// TwinCAT 3 PLC project TcSequencer
// Title: TcSequencer
// Company: Loupe
// ProjectVersion: 0.0.5
// ProgramVersion: 3.1.4024.0
// libraries:
//   Tc2_Standard, * (Beckhoff Automation GmbH)
//   Tc2_System, * (Beckhoff Automation GmbH)
//   Tc3_Module, * (Beckhoff Automation GmbH)
//   TcCommando, * (Loupe)
//   TcPluginFramework, * (Loupe)
//   TcUnit, * (www.tcunit.org)
// project tree:
//   DUTs/ SequenceCommand.TcDUT, SequenceType.TcDUT, SEQUENCE_STEP.TcTLEO
//   Example/ ExampleProg1.TcPOU, ExampleSeq1.TcPOU, IMOCK_EM.TcIO, Mock_EM.TcPOU
//   Interfaces/ ISequence.TcIO, IStepManager.TcIO
//   / PlcTask.TcTTO
//   POUs/ Sequencer.TcPOU, StepManagerBasic.TcPOU
//   Test/ Sequencer_Test.TcPOU, StepManagerBasic_Test.TcPOU, TESTPRG.TcPOU
// real-time tasks:
//   TASK PlcTask: cycle T#10ms, priority 20, ADS port 350

CONFIGURATION TcSequencer
    RESOURCE PLC ON TwinCAT3
        TASK PlcTask(INTERVAL := T#10ms, PRIORITY := 20);
        PROGRAM TESTPRG WITH PlcTask : TESTPRG;
        PROGRAM ExampleProg1 WITH PlcTask : ExampleProg1;
    END_RESOURCE
END_CONFIGURATION

// ---- DUTs/SequenceCommand.TcDUT
TYPE SequenceCommand :
STRUCT
	Start : PLCopenCommand;
	Stop : PLCopenCommand;
END_STRUCT
END_TYPE

// ---- DUTs/SequenceType.TcDUT
TYPE
    SequenceType :
    STRUCT
        startStep : ENUM; //The step when doStep was called
        currentStep : ENUM;
        lastRequestNumber : DINT;

        onEntry : BOOL;
        onExit : BOOL;

        statusChecked : BOOL;
        isDone : BOOL;
        isAbort : BOOL;
        isError : BOOL;

        errorHandled : BOOL;

    END_STRUCT
END_TYPE

// ---- DUTs/SEQUENCE_STEP.TcTLEO
{attribute 'qualified_only'}
TYPE SEQUENCE_STEP :
(
	STEP_ERROR := -3,
	NO_STEP_CHANGE := -2,
	NO_STEP := -1,
	IDLE_STEP := 0,
	START_STEP := 1
);
END_TYPE
//  STEP_ERROR = '-3'
//  NO_STEP_CHANGE = '-2'
//  NO_STEP = '-1'

// ---- Example/IMOCK_EM.TcIO
INTERFACE IMOCK_EM


METHOD MoveDown : BOOL
VAR_INPUT
  Status : IPLCopenCall;
END_VAR
END_METHOD


METHOD MoveUp : BOOL
VAR_INPUT
  Status : IPLCopenCall;
END_VAR
END_METHOD

END_INTERFACE

// ---- Interfaces/ISequence.TcIO
INTERFACE ISequence
// Copyright (c) 2024 Loupe (https://loupe.team), provided under the MIT License.

{attribute 'monitoring' := 'call'}
PROPERTY CurrentStep : ENUM
GET
END_GET
END_PROPERTY

METHOD DoStep : ENUM
VAR
END_VAR
END_METHOD

METHOD OnAbort : BOOL
VAR_INPUT
    nextStep : ENUM;
END_VAR
END_METHOD

METHOD OnEntry : BOOL
VAR_INPUT
END_VAR
END_METHOD

METHOD OnError : BOOL
VAR_INPUT
    nextStep : ENUM;
END_VAR
END_METHOD

METHOD OnExit : BOOL
VAR_INPUT
END_VAR
END_METHOD

METHOD OnFailure : BOOL
VAR_INPUT
    nextStep : ENUM;
END_VAR
END_METHOD

METHOD OnSuccess : BOOL
VAR_INPUT
    nextStep : ENUM;
END_VAR
END_METHOD

METHOD RequestStep : BOOL
VAR_INPUT
    nextStep : ENUM;
END_VAR
END_METHOD

METHOD RequestStepClear : BOOL
VAR_INPUT
    nextStep : ENUM;
END_VAR
END_METHOD

METHOD SequenceAbort : BOOL
VAR_INPUT
    ErrorCode : DINT;
    ErrorMessage : STRING;
END_VAR
END_METHOD

METHOD SequenceComplete : BOOL
VAR_INPUT
END_VAR
END_METHOD

METHOD SequenceError : BOOL
VAR_INPUT
    ErrorCode : INT;
    ErrorMessage : STRING;
END_VAR
END_METHOD

METHOD SetStepManager : BOOL
VAR_INPUT
	manager : IStepManager;
END_VAR
END_METHOD

METHOD StartSequence : BOOL
VAR_INPUT
	Status : IPLCopenCaller;
END_VAR
END_METHOD

END_INTERFACE

// ---- Interfaces/IStepManager.TcIO
INTERFACE IStepManager
// Copyright (c) 2024 Loupe (https://loupe.team), provided under the MIT License.

PROPERTY CurrentStepImpl : ENUM
GET
END_GET
END_PROPERTY

PROPERTY RequestNumberImpl : DINT
GET
END_GET
END_PROPERTY

METHOD RequestStepImpl : BOOL
VAR_INPUT
    nextStep : ENUM;
END_VAR
END_METHOD

METHOD ResetImpl : BOOL
VAR_INPUT
END_VAR
END_METHOD

METHOD SequenceCompleteImpl : BOOL
VAR_INPUT
END_VAR
END_METHOD

METHOD SequenceErrorImpl : BOOL
VAR_INPUT
    ErrorCode : INT;
    ErrorMessage : STRING;
END_VAR
END_METHOD

END_INTERFACE

// ---- Test/TESTPRG.TcPOU
{attribute 'no-analysis'}
PROGRAM TESTPRG
VAR
    sequencerTest : Sequencer_Test;
    stepManagerTest : StepManagerBasic_Test;
END_VAR

// Copyright (c) 2024 Loupe (https://loupe.team), provided under the MIT License.

TcUnit.RUN();

END_PROGRAM

// ---- Test/Sequencer_Test.TcPOU
FUNCTION_BLOCK Sequencer_Test EXTENDS FB_TestSuite
VAR_INPUT
END_VAR
VAR_OUTPUT
END_VAR
VAR
END_VAR

// Copyright (c) 2024 Loupe (https://loupe.team), provided under the MIT License.

OnAbort();
OnEntry();
CurrentAndRequestStep();

{attribute 'no-analysis'}
METHOD CurrentAndRequestStep
VAR
    sequencer : Sequencer(0);
    Command : PLCopenCommand();
    step : UDINT;
END_VAR
// Copyright (c) 2024 Loupe (https://loupe.team), provided under the MIT License.

(*STweep.Disable*)

TEST('CurrentAndRequestStep');
	AssertEquals_UDINT(Expected := 0, Actual := sequencer.CurrentStep, Message := 'Current step shall default to 0');
	
	step := 2;
	sequencer.RequestStep(step);
	AssertEquals_UDINT(Expected := step, Actual := sequencer.CurrentStep, Message := 'Current step expected to be updated');
	
	step := 3;
	sequencer.RequestStepClear(step);
	AssertEquals_UDINT(Expected := step, Actual := sequencer.CurrentStep, Message := 'Current step expected to be updated');
TEST_FINISHED();
END_METHOD

{attribute 'no-analysis'}
METHOD OnAbort
VAR
    sequencer : Sequencer(0);
    outputVal : BOOL;
	Command : PLCopenCommand;
END_VAR
// Copyright (c) 2024 Loupe (https://loupe.team), provided under the MIT License.

(*STweep.Disable*)

TEST('SequenceOnAbort');
	sequencer.RequestStep(1);
	sequencer.DoStep();
	sequencer.Start(Command);
	Command.Execute := TRUE;
	IF sequencer.OnAbort(-1) THEN
		outputVal := sequencer.SequenceAbort(1, 'Command aborted');
	END_IF
	AssertTrue(Condition := outputVal, Message := 'Abort should be true');
TEST_FINISHED();
END_METHOD

{attribute 'no-analysis'}
METHOD OnEntry
VAR_INPUT
END_VAR

VAR
    sequencer : Sequencer(0);
    outputVal : BOOL;
END_VAR
// Copyright (c) 2024 Loupe (https://loupe.team), provided under the MIT License.

(*STweep.Disable*)

TEST('OnEntry');
	
	sequencer.StartSequence(0);
	sequencer.DoStep();
	AssertTrue(Condition := sequencer.onEntry(), Message := 'onEntry should evaluate TRUE on first pass through a new step');
	sequencer.DoStep();
	AssertFalse(Condition := sequencer.onEntry(), Message := 'onEntry should evaluate FALSE on second pass');
	
TEST_FINISHED();
END_METHOD

{attribute 'no-analysis'}
{attribute 'no-analysis'}
METHOD OnError
VAR
    sequencer : Sequencer(0);
    outputVal : BOOL;
	Command : PLCopenCommand;
END_VAR
// Copyright (c) 2024 Loupe (https://loupe.team), provided under the MIT License.

(*STweep.Disable*)

TEST('SequenceOnError');
	sequencer.RequestStep(1);
	sequencer.DoStep();
	sequencer.Start(Command);
	Command.Errored(1);
	IF sequencer.OnError(1) THEN
		outputVal := sequencer.SequenceError(0, 'Test Error');
	END_IF

	AssertTrue(Condition := outputVal, Message := 'Error should be true');
TEST_FINISHED();
END_METHOD

{attribute 'no-analysis'}
METHOD OnSuccess
VAR_INPUT
    sequencer : Sequencer(0);
END_VAR
// Copyright (c) 2024 Loupe (https://loupe.team), provided under the MIT License.

(*STweep.Disable*)

TEST('OnSuccess');

	//sequencer._sequence.activeTasks
	// next step negative
	//sequencer.setNextStep(-1);
	//sequencer.onSuccess(-1);
	
	// next step >= 0


TEST_FINISHED();
END_METHOD

{attribute 'no-analysis'}
METHOD Start
VAR
    sequencer : Sequencer(0);
    output : BOOL;
END_VAR
// Copyright (c) 2024 Loupe (https://loupe.team), provided under the MIT License.

(*STweep.Disable*)

TEST('Start');
	// activeTasks.Start) = 0
	// TODO
	
	//output := sequencer._sequence.startStep
	
	
TEST_FINISHED();
END_METHOD

END_FUNCTION_BLOCK

// ---- POUs/Sequencer.TcPOU
FUNCTION_BLOCK Sequencer IMPLEMENTS ISequence, IPlugin, IPLCopenCall
VAR_INPUT	
  startStep : ENUM;
  Command : SequenceCommand;
END_VAR
VAR
  _sequence : SequenceType;
  _activeTasks : PLCopenCallGroup;
  _stepHandler : IStepManager;
  _baseManager : StepManagerBasic;
END_VAR

// Copyright (c) 2024 Loupe (https://loupe.team), provided under the MIT License.


METHOD PRIVATE CheckStatus : BOOL

// Copyright (c) 2024 Loupe (https://loupe.team), provided under the MIT License.

IF NOT _sequence.statusChecked THEN
  _sequence.statusChecked := TRUE;
  // Cache the abort so there's a consistent status for the whole state
  _sequence.isError := _activeTasks.Error;
  _sequence.isAbort := _activeTasks.CommandAborted;
  _sequence.isDone := _activeTasks.Done;
END_IF
END_METHOD


{attribute 'monitoring' := 'call'}
PROPERTY CurrentStep : ENUM
GET
// Copyright (c) 2024 Loupe (https://loupe.team), provided under the MIT License.

CurrentStep := _stepHandler.CurrentStepImpl;
END_GET
END_PROPERTY


METHOD DoStep : ENUM
VAR
END_VAR
// Copyright (c) 2024 Loupe (https://loupe.team), provided under the MIT License.


IF Command.Start.Consume THEN
  _stepHandler.RequestStepImpl(startStep);
END_IF

_sequence.currentStep := _stepHandler.CurrentStepImpl;

//If the current step has changed,
//	Set the flag for onEntry()
IF _stepHandler.RequestNumberImpl <> _sequence.lastRequestNumber THEN

  _sequence.lastRequestNumber := _stepHandler.RequestNumberImpl;
  _sequence.onEntry := TRUE;
  _sequence.onExit := FALSE;
ELSE
  _sequence.onEntry := FALSE;
END_IF

//The start step is used to detect if the 
_sequence.startStep := _sequence.currentStep;

//Mark that we haven't checked the status yet, 
//	This is to ensure we don't have inconsitent onCalls
_sequence.statusChecked := FALSE;
_sequence.errorHandled := FALSE;

IF _sequence.onExit THEN
  DoStep := SEQUENCE_STEP.NO_STEP;
ELSE
  //Return the state
  DoStep := _sequence.currentStep;
END_IF
END_METHOD


METHOD FB_init : BOOL
VAR_INPUT
  bInitRetains : BOOL; // if TRUE, the retain variables are initialized (warm start / cold start)
  bInCopyCode : BOOL; // if TRUE, the instance afterwards gets moved into the copy code (online change)
  stepHandler : IStepManager;
END_VAR

// Copyright (c) 2024 Loupe (https://loupe.team), provided under the MIT License.

IF stepHandler = 0 THEN
  _stepHandler := _baseManager;
ELSE
  _stepHandler := stepHandler;
END_IF
END_METHOD


PROPERTY IsAbort : BOOL
GET

// Copyright (c) 2024 Loupe (https://loupe.team), provided under the MIT License.

CheckStatus();
IsAbort := _sequence.isAbort;
END_GET
END_PROPERTY


PROPERTY IsDone : BOOL
GET

// Copyright (c) 2024 Loupe (https://loupe.team), provided under the MIT License.

CheckStatus();
IsDone := _sequence.isDone;
END_GET
END_PROPERTY


PROPERTY IsError : BOOL
GET

// Copyright (c) 2024 Loupe (https://loupe.team), provided under the MIT License.

CheckStatus();
IsError := _sequence.isError;
END_GET
END_PROPERTY


METHOD OnAbort : BOOL
VAR_INPUT
  nextStep : ENUM;
END_VAR

// Copyright (c) 2024 Loupe (https://loupe.team), provided under the MIT License.

// Check all of the status to see if we are aborting

IF IsAbort THEN

  IF nextStep >= 0 THEN
    LogMessage(1, 'Step Abort');
    _sequence.errorHandled := TRUE;
    setNextStep(nextStep);
  END_IF

  OnAbort := TRUE;
ELSE
  OnAbort := FALSE;
END_IF
END_METHOD


METHOD OnEntry : BOOL

// Copyright (c) 2024 Loupe (https://loupe.team), provided under the MIT License.

//If the current step has since the doStep
OnEntry := _sequence.onEntry;
END_METHOD


METHOD OnError : BOOL
VAR_INPUT
  nextStep : ENUM;
END_VAR

// Copyright (c) 2024 Loupe (https://loupe.team), provided under the MIT License.

IF IsError THEN
  IF nextStep >= 0 THEN
    LogMessage(1, 'Step Abort');
    _sequence.errorHandled := TRUE;
    setNextStep(nextStep);
  END_IF

  OnError := TRUE;
ELSE
  OnError := FALSE;
END_IF
END_METHOD

METHOD OnExit : BOOL

// Copyright (c) 2024 Loupe (https://loupe.team), provided under the MIT License.

//If the current step has since the doStep
OnExit := _sequence.onExit;
END_METHOD


METHOD OnFailure : BOOL
VAR_INPUT
  nextStep : ENUM;
END_VAR

// Copyright (c) 2024 Loupe (https://loupe.team), provided under the MIT License.

IF IsAbort OR IsError THEN
  //On failure will not set the step if a more specific handler already set the step
  IF _sequence.errorHandled = FALSE AND nextStep >= 0 THEN
    LogMessage(1, 'Step Failure');
    setNextStep(nextStep);
  END_IF

  OnFailure := TRUE;
ELSE
  OnFailure := FALSE;
END_IF
END_METHOD


METHOD OnSuccess : BOOL
VAR_INPUT
  nextStep : ENUM;
END_VAR

// Copyright (c) 2024 Loupe (https://loupe.team), provided under the MIT License.

IF IsDone THEN
  IF nextStep >= 0 THEN
    LogMessage(1, 'Step Success');
    setNextStep(nextStep);
  END_IF

  OnSuccess := TRUE;
ELSE
  OnSuccess := FALSE;
END_IF
END_METHOD


METHOD RequestStep : BOOL
VAR_INPUT
  nextStep : ENUM;
END_VAR
// Copyright (c) 2024 Loupe (https://loupe.team), provided under the MIT License.

_stepHandler.RequestStepImpl(nextStep);
_sequence.onExit := TRUE;
END_METHOD


METHOD RequestStepClear : BOOL
VAR_INPUT
  nextStep : ENUM;
END_VAR

// Copyright (c) 2024 Loupe (https://loupe.team), provided under the MIT License.

RequestStep(nextStep);
_activeTasks.ResetStatus();
END_METHOD


METHOD Run : BOOL

// Copyright (c) 2024 Loupe (https://loupe.team), provided under the MIT License.

THIS^();
END_METHOD


METHOD SequenceAbort : BOOL
VAR_INPUT
  ErrorCode : DINT;
  ErrorMessage : STRING;
END_VAR
// Copyright (c) 2024 Loupe (https://loupe.team), provided under the MIT License.

_stepHandler.SequenceErrorImpl(DINT_TO_INT(ErrorCode), ErrorMessage);
_activeTasks.ResetStatus();
_sequence.onExit := TRUE;
Command.Start.Aborted();
SequenceAbort := TRUE;
END_METHOD


METHOD SequenceComplete : BOOL
VAR_INPUT
END_VAR

// Copyright (c) 2024 Loupe (https://loupe.team), provided under the MIT License.

_stepHandler.SequenceCompleteImpl();
_activeTasks.ResetStatus();
_sequence.onExit := TRUE;
Command.Start.Finished();
SequenceComplete := TRUE;
END_METHOD


METHOD SequenceError : BOOL
VAR_INPUT
  ErrorCode : INT;
  ErrorMessage : STRING;
END_VAR

// Copyright (c) 2024 Loupe (https://loupe.team), provided under the MIT License.

_stepHandler.SequenceErrorImpl(ErrorCode, ErrorMessage);
_activeTasks.ResetStatus();
_sequence.onExit := TRUE;
Command.Start.Errored(ErrorCode);
SequenceError := TRUE;
END_METHOD


METHOD PROTECTED SetNextStep
VAR_INPUT
  nextStep : ENUM;
END_VAR
// Copyright (c) 2024 Loupe (https://loupe.team), provided under the MIT License.

_stepHandler.RequestStepImpl(nextStep);
END_METHOD

METHOD SetStepManager : BOOL
VAR_INPUT
	manager	: IStepManager;
END_VAR
_stepHandler := manager;
END_METHOD


METHOD Start : PLCopenStatusBase
VAR_INPUT
  Command : IPLCopenCommand;
END_VAR
VAR
	_status : PLCopenStatusBase;
END_VAR

// Copyright (c) 2024 Loupe (https://loupe.team), provided under the MIT License.
_status := _activeTasks.Start(Command);
IF  _status <> PLCopenStatusBase.BUSY THEN
  // TODO: All out of commands.. Throw an error
  sequenceError(10000, 'Too Many Commands in 1 step');
END_IF
Start := _status;
END_METHOD


METHOD StartSequence : BOOL
VAR_INPUT
	Status : IPLCopenCaller;
END_VAR

// Copyright (c) 2024 Loupe (https://loupe.team), provided under the MIT License.
IF Status <> 0 THEN
	Status.Start(Command.Start);
ELSE
	Command.Start.Execute := TRUE;
END_IF
END_METHOD

END_FUNCTION_BLOCK

// ---- POUs/StepManagerBasic.TcPOU
{attribute 'enable_dynamic_creation'}
FUNCTION_BLOCK StepManagerBasic IMPLEMENTS IStepManager
VAR
    _currentStep : ENUM;
    _requestNumber : DINT;
END_VAR

// Copyright (c) 2024 Loupe (https://loupe.team), provided under the MIT License.

PROPERTY CurrentStepImpl : ENUM
GET
// Copyright (c) 2024 Loupe (https://loupe.team), provided under the MIT License.

CurrentStepImpl := _CurrentStep;
END_GET
END_PROPERTY

{warning 'add property implementation'}
PROPERTY RequestNumberImpl : DINT
GET
// Copyright (c) 2024 Loupe (https://loupe.team), provided under the MIT License.

RequestNumberImpl := _requestNumber;
END_GET
END_PROPERTY

METHOD RequestStepImpl : BOOL
VAR_INPUT
    nextStep : ENUM;
END_VAR
// Copyright (c) 2024 Loupe (https://loupe.team), provided under the MIT License.

_requestNumber := _requestNumber + 1;
_currentStep := nextStep;
END_METHOD

METHOD ResetImpl : BOOL
// Copyright (c) 2024 Loupe (https://loupe.team), provided under the MIT License.

_currentStep := SEQUENCE_STEP.NO_STEP;
END_METHOD

METHOD SequenceCompleteImpl : BOOL
// Copyright (c) 2024 Loupe (https://loupe.team), provided under the MIT License.

_requestNumber := _requestNumber + 1;
_currentStep := SEQUENCE_STEP.NO_STEP;
END_METHOD

METHOD SequenceErrorImpl : BOOL
VAR_INPUT
    ErrorCode : INT;
    ErrorMessage : STRING;
END_VAR
// Copyright (c) 2024 Loupe (https://loupe.team), provided under the MIT License.

_requestNumber := _requestNumber + 1;
_currentStep := SEQUENCE_STEP.NO_STEP;
END_METHOD

END_FUNCTION_BLOCK

// ---- Test/StepManagerBasic_Test.TcPOU
{attribute 'no-analysis'}
FUNCTION_BLOCK StepManagerBasic_Test EXTENDS FB_TestSuite
VAR_INPUT
END_VAR
VAR_OUTPUT
END_VAR
VAR
END_VAR

// Copyright (c) 2024 Loupe (https://loupe.team), provided under the MIT License.

RequestStep();
Reset();

METHOD RequestStep
VAR
    stepManager : StepManagerBasic();
END_VAR
// Copyright (c) 2024 Loupe (https://loupe.team), provided under the MIT License.

(*STweep.Disable*)

TEST('RequestStep');
	stepManager.RequestStepImpl(2);
	AssertEquals_UDINT(Expected := 2, Actual := stepManager.CurrentStepImpl, 'Current Step shall be requested step');
TEST_FINISHED();
END_METHOD

METHOD Reset
VAR
    stepManager : StepManagerBasic();
END_VAR
// Copyright (c) 2024 Loupe (https://loupe.team), provided under the MIT License.

(*STweep.Disable*)

TEST('Reset');
	stepManager.RequestStepImpl(20);
	AssertEquals_UDINT(Expected := 20, Actual := stepManager.CurrentStepImpl, 'Confirm current step is not default');
	
	stepManager.ResetImpl();
	AssertEquals_UDINT(Expected := SEQUENCE_STEP.NO_STEP, Actual := stepManager.CurrentStepImpl, 'Reset should have put current step back to default');
TEST_FINISHED();
END_METHOD

END_FUNCTION_BLOCK

// ---- Example/ExampleProg1.TcPOU
PROGRAM ExampleProg1
VAR

	Cylinder1 : Mock_EM := (TimeUp:= T#3S, TimeDown:= T#3S);		
	Cylinder2 : Mock_EM := (TimeUp:= T#1S, TimeDown:= T#1S);
	Cylinder3 : Mock_EM := (TimeUp:= T#8S, TimeDown:= T#1S);
	Seq1 :	ExampleSeq1(0) := (em1:=Cylinder1, em2:=Cylinder2, em3:=Cylinder3);
END_VAR

Cylinder1();
Cylinder2();
Cylinder3();

Seq1();

END_PROGRAM

// ---- Example/Mock_EM.TcPOU

FUNCTION_BLOCK Mock_EM IMPLEMENTS IMOCK_EM
VAR_INPUT
  TimeUp : TIME;
  TimeDown : TIME;
END_VAR
VAR
  _MoveUp : PLCopenCommand;
  _MoveDown : PLCopenCommand;
  _HeightGroup : PLCopenExclusiveGroup := (commands := [_MoveUp, _MoveDown, 18(0)]); 
  t : TON;
  Up : BOOL;
  Down : BOOL;
  Up_ : BOOL;
END_VAR


IF _MoveDown.Consume THEN

  t(IN := FALSE);
  t(IN := TRUE, PT := TimeDown);
  Up_ := FALSE;
  Up := FALSE;
  Down := FALSE;

END_IF

IF _MoveUp.Consume THEN

  t(IN := FALSE);
  t(IN := TRUE, PT := TimeUp);
  Up_ := TRUE;
  Up := FALSE;
  Down := FALSE;

END_IF

t();

IF t.Q THEN

  t(IN := FALSE);

  IF Up_ THEN
    Up := TRUE;
	_MoveUp.Finished();
  ELSE
    Down := TRUE;
	_MoveDown.Finished();
  END_IF

END_IF


METHOD MoveDown : BOOL
VAR_INPUT
  Status : IPLCopenCall;
END_VAR

Status.Start(_MoveDown);
END_METHOD


METHOD MoveUp : BOOL
VAR_INPUT
  Status : IPLCopenCall;
END_VAR

Status.Start(_MoveUp);
END_METHOD

END_FUNCTION_BLOCK

// ---- Example/ExampleSeq1.TcPOU
FUNCTION_BLOCK ExampleSeq1 EXTENDS Sequencer
VAR_INPUT
	em1 : IMOCK_EM;
	em2 : IMOCK_EM;
	em3 : IMOCK_EM;
END_VAR

CASE DoStep() OF

	0:
		IF OnEntry() THEN
			RequestStep( 1 );			
		END_IF

	1: 
		IF OnEntry() THEN
			em1.MoveDown(THIS^);
		END_IF	

		OnSuccess(2);
	2:

		IF OnEntry() THEN
			em1.MoveUp(THIS^);
			em2.MoveUp(THIS^);
			em3.MoveUp(THIS^);			
		END_IF
	
		OnSuccess(3);
		
	3:		
				
		IF OnEntry() THEN
			em1.MoveDown(THIS^);
			em2.MoveDown(THIS^);
			em3.MoveUp(THIS^);			
		END_IF
	
		
		IF OnSuccess(-1) THEN

			SequenceComplete();			

		END_IF
		
END_CASE

IF OnError(-1) THEN
	SequenceError(-1, 'General error');
END_IF

END_FUNCTION_BLOCK
